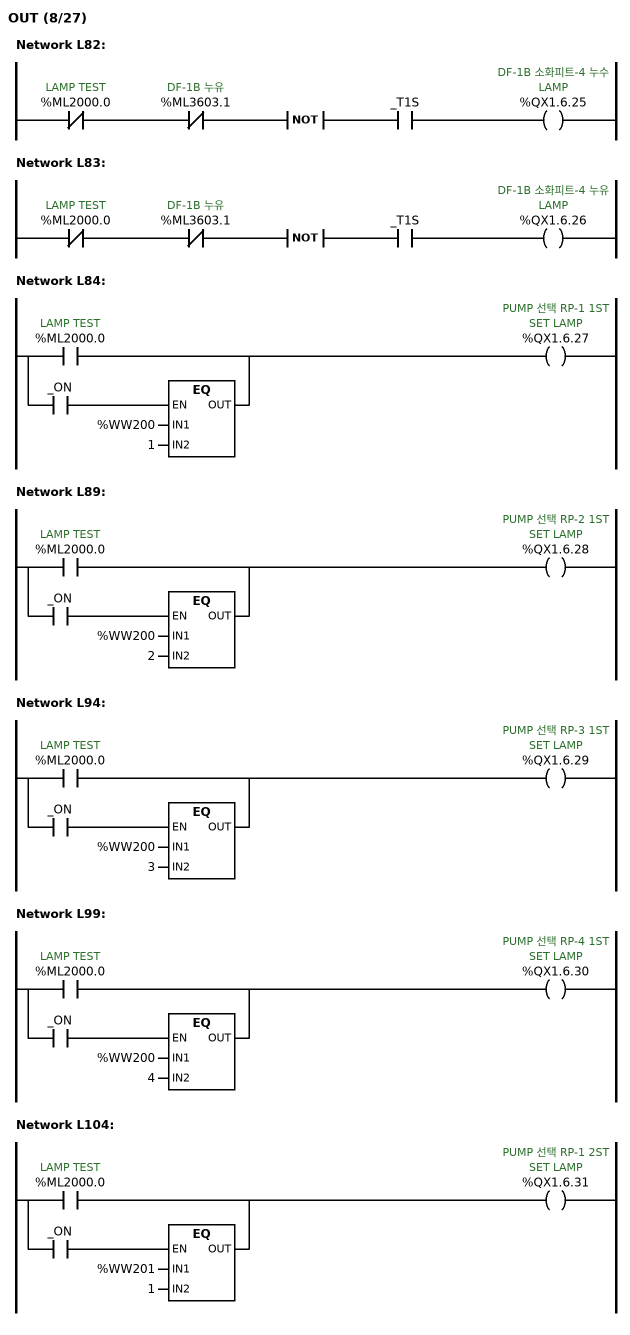
(* Rung L82 *)
%QX1.6.25 := NOT (NOT %ML2000.0 AND NOT %ML3603.1) AND _T1S;
(* Rung L83 *)
%QX1.6.26 := NOT (NOT %ML2000.0 AND NOT %ML3603.1) AND _T1S;
(* Rung L84 *)
IF _ON THEN _t1 := %WW200 = 1; END_IF;
%QX1.6.27 := %ML2000.0 OR _t1;
(* Rung L89 *)
IF _ON THEN _t2 := %WW200 = 2; END_IF;
%QX1.6.28 := %ML2000.0 OR _t2;
(* Rung L94 *)
IF _ON THEN _t3 := %WW200 = 3; END_IF;
%QX1.6.29 := %ML2000.0 OR _t3;
(* Rung L99 *)
IF _ON THEN _t4 := %WW200 = 4; END_IF;
%QX1.6.30 := %ML2000.0 OR _t4;
(* Rung L104 *)
IF _ON THEN _t5 := %WW201 = 1; END_IF;
%QX1.6.31 := %ML2000.0 OR _t5;

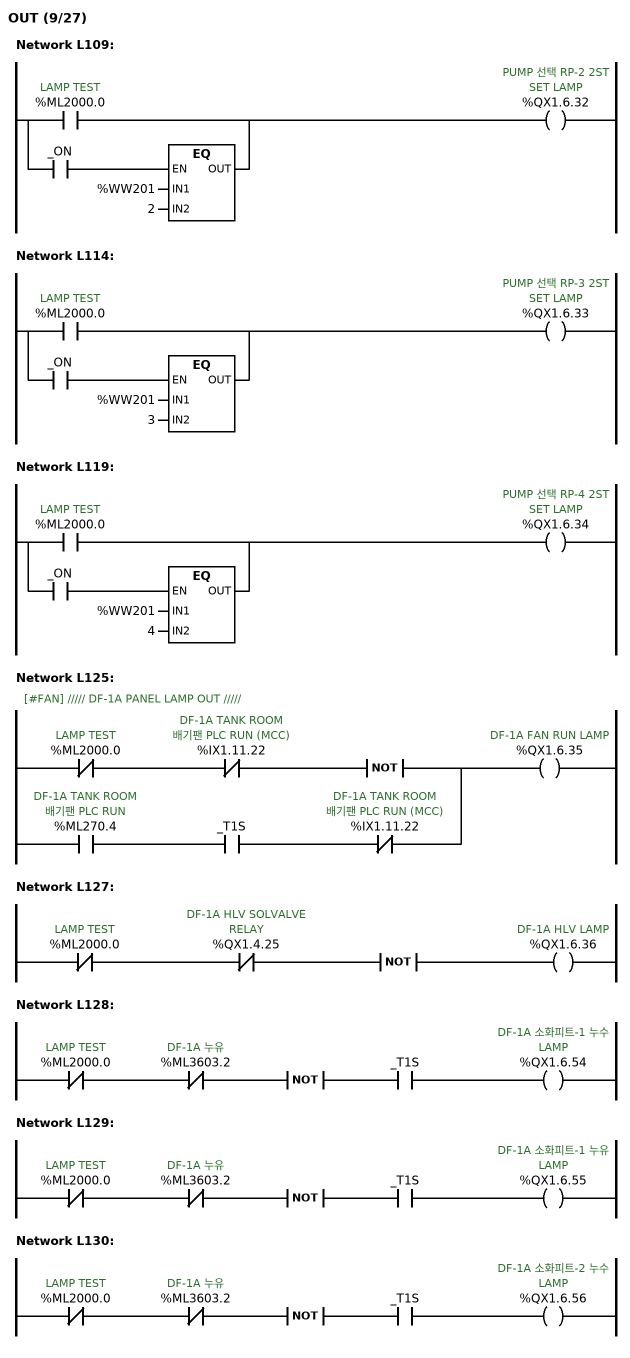
(* Rung L109 *)
IF _ON THEN _t6 := %WW201 = 2; END_IF;
%QX1.6.32 := %ML2000.0 OR _t6;
(* Rung L114 *)
IF _ON THEN _t7 := %WW201 = 3; END_IF;
%QX1.6.33 := %ML2000.0 OR _t7;
(* Rung L119 *)
IF _ON THEN _t8 := %WW201 = 4; END_IF;
%QX1.6.34 := %ML2000.0 OR _t8;
(* [#FAN] ///// DF-1A PANEL LAMP OUT ///// *)
(* Rung L125 *)
%QX1.6.35 := NOT (NOT %ML2000.0 AND NOT %IX1.11.22) OR (%ML270.4 AND _T1S AND NOT %IX1.11.22);
(* Rung L127 *)
%QX1.6.36 := NOT (NOT %ML2000.0 AND NOT %QX1.4.25);
(* Rung L128 *)
%QX1.6.54 := NOT (NOT %ML2000.0 AND NOT %ML3603.2) AND _T1S;
(* Rung L129 *)
%QX1.6.55 := NOT (NOT %ML2000.0 AND NOT %ML3603.2) AND _T1S;
(* Rung L130 *)
%QX1.6.56 := NOT (NOT %ML2000.0 AND NOT %ML3603.2) AND _T1S;

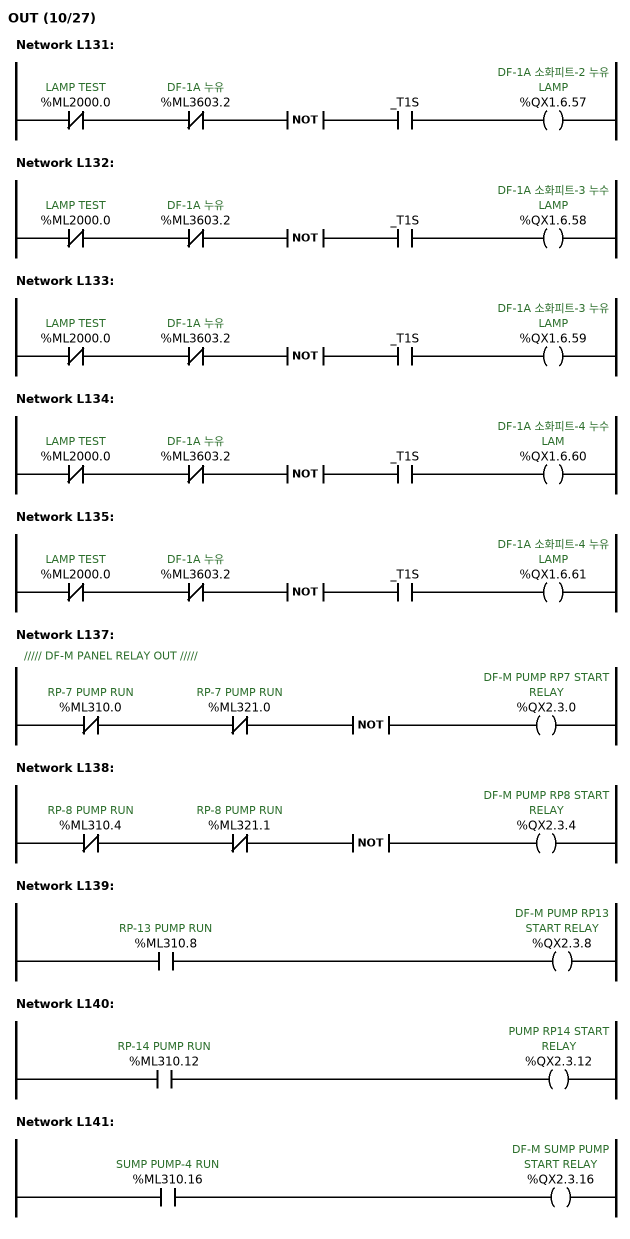
(* Rung L131 *)
%QX1.6.57 := NOT (NOT %ML2000.0 AND NOT %ML3603.2) AND _T1S;
(* Rung L132 *)
%QX1.6.58 := NOT (NOT %ML2000.0 AND NOT %ML3603.2) AND _T1S;
(* Rung L133 *)
%QX1.6.59 := NOT (NOT %ML2000.0 AND NOT %ML3603.2) AND _T1S;
(* Rung L134 *)
%QX1.6.60 := NOT (NOT %ML2000.0 AND NOT %ML3603.2) AND _T1S;
(* Rung L135 *)
%QX1.6.61 := NOT (NOT %ML2000.0 AND NOT %ML3603.2) AND _T1S;
(* ///// DF-M PANEL RELAY OUT ///// *)
(* Rung L137 *)
%QX2.3.0 := NOT (NOT %ML310.0 AND NOT %ML321.0);
(* Rung L138 *)
%QX2.3.4 := NOT (NOT %ML310.4 AND NOT %ML321.1);
(* Rung L139 *)
%QX2.3.8 := %ML310.8;
(* Rung L140 *)
%QX2.3.12 := %ML310.12;
(* Rung L141 *)
%QX2.3.16 := %ML310.16;

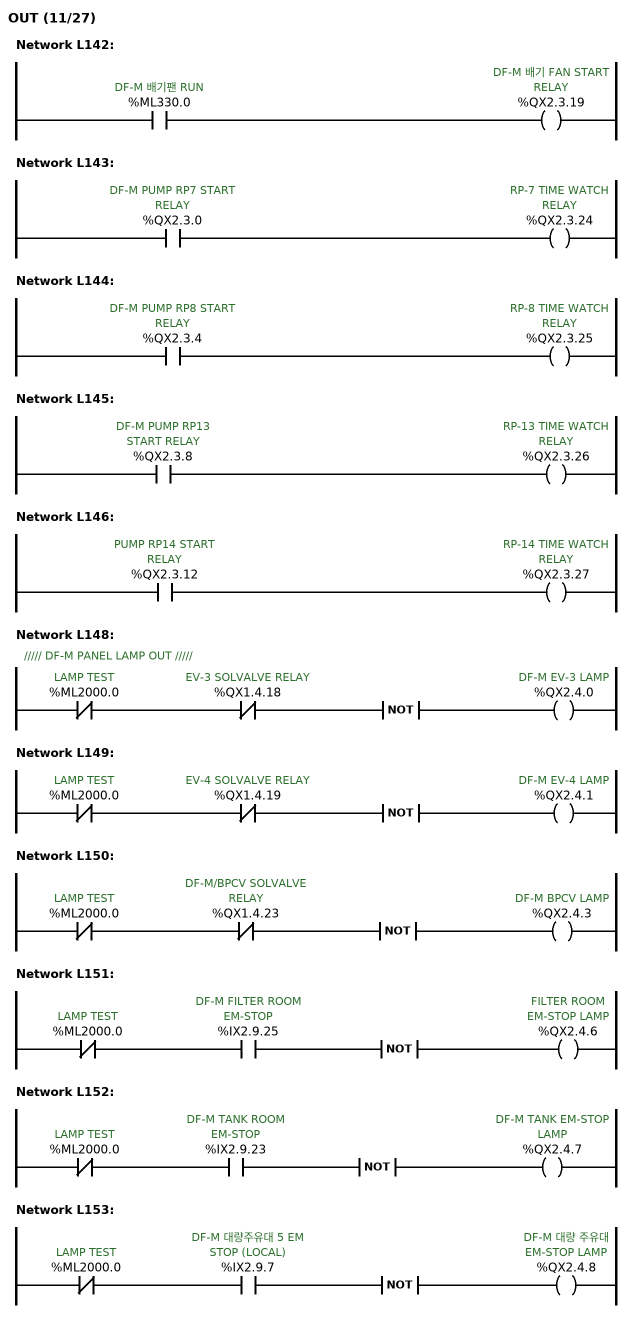
(* Rung L142 *)
%QX2.3.19 := %ML330.0;
(* Rung L143 *)
%QX2.3.24 := %QX2.3.0;
(* Rung L144 *)
%QX2.3.25 := %QX2.3.4;
(* Rung L145 *)
%QX2.3.26 := %QX2.3.8;
(* Rung L146 *)
%QX2.3.27 := %QX2.3.12;
(* ///// DF-M PANEL LAMP OUT ///// *)
(* Rung L148 *)
%QX2.4.0 := NOT (NOT %ML2000.0 AND NOT %QX1.4.18);
(* Rung L149 *)
%QX2.4.1 := NOT (NOT %ML2000.0 AND NOT %QX1.4.19);
(* Rung L150 *)
%QX2.4.3 := NOT (NOT %ML2000.0 AND NOT %QX1.4.23);
(* Rung L151 *)
%QX2.4.6 := NOT (NOT %ML2000.0 AND %IX2.9.25);
(* Rung L152 *)
%QX2.4.7 := NOT (NOT %ML2000.0 AND %IX2.9.23);
(* Rung L153 *)
%QX2.4.8 := NOT (NOT %ML2000.0 AND %IX2.9.7);

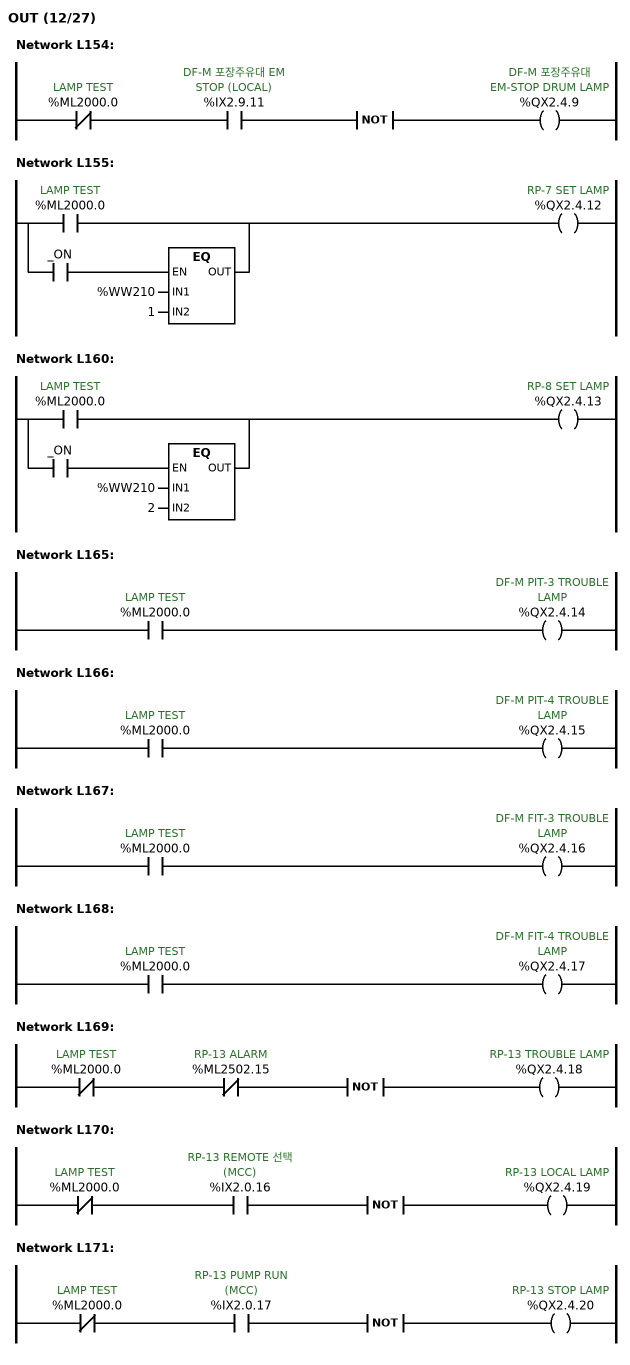
(* Rung L154 *)
%QX2.4.9 := NOT (NOT %ML2000.0 AND %IX2.9.11);
(* Rung L155 *)
IF _ON THEN _t9 := %WW210 = 1; END_IF;
%QX2.4.12 := %ML2000.0 OR _t9;
(* Rung L160 *)
IF _ON THEN _t10 := %WW210 = 2; END_IF;
%QX2.4.13 := %ML2000.0 OR _t10;
(* Rung L165 *)
%QX2.4.14 := %ML2000.0;
(* Rung L166 *)
%QX2.4.15 := %ML2000.0;
(* Rung L167 *)
%QX2.4.16 := %ML2000.0;
(* Rung L168 *)
%QX2.4.17 := %ML2000.0;
(* Rung L169 *)
%QX2.4.18 := NOT (NOT %ML2000.0 AND NOT %ML2502.15);
(* Rung L170 *)
%QX2.4.19 := NOT (NOT %ML2000.0 AND %IX2.0.16);
(* Rung L171 *)
%QX2.4.20 := NOT (NOT %ML2000.0 AND %IX2.0.17);

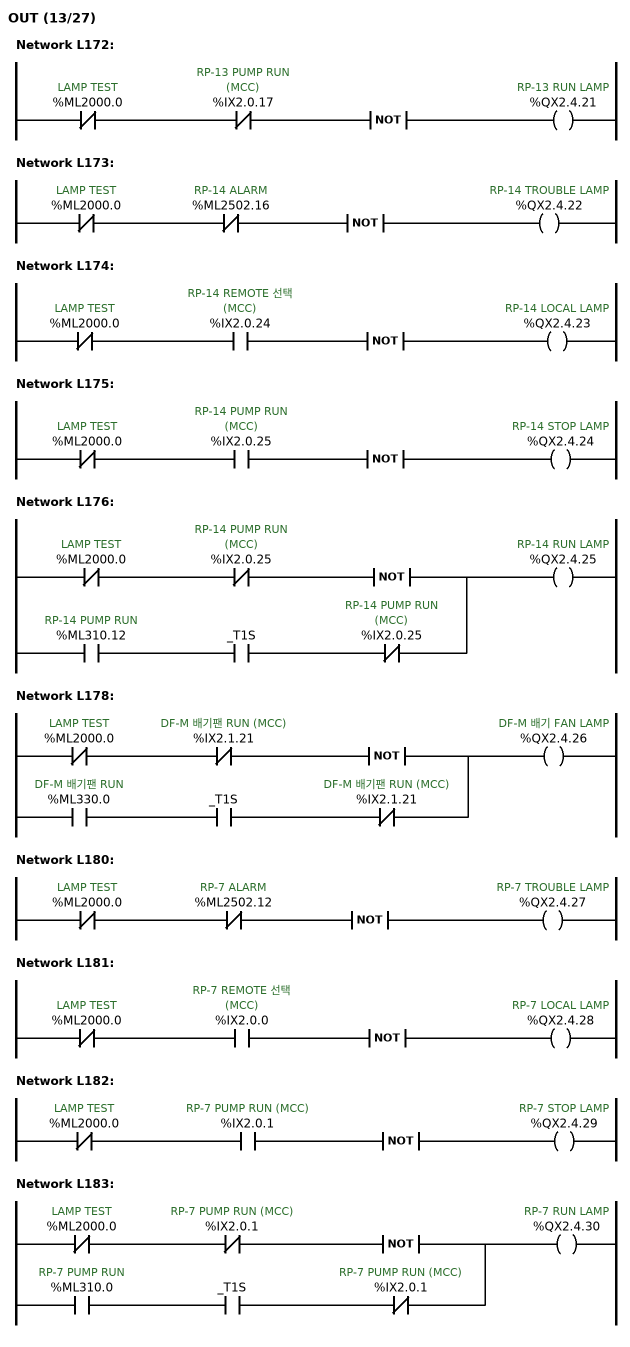
(* Rung L172 *)
%QX2.4.21 := NOT (NOT %ML2000.0 AND NOT %IX2.0.17);
(* Rung L173 *)
%QX2.4.22 := NOT (NOT %ML2000.0 AND NOT %ML2502.16);
(* Rung L174 *)
%QX2.4.23 := NOT (NOT %ML2000.0 AND %IX2.0.24);
(* Rung L175 *)
%QX2.4.24 := NOT (NOT %ML2000.0 AND %IX2.0.25);
(* Rung L176 *)
%QX2.4.25 := NOT (NOT %ML2000.0 AND NOT %IX2.0.25) OR (%ML310.12 AND _T1S AND NOT %IX2.0.25);
(* Rung L178 *)
%QX2.4.26 := NOT (NOT %ML2000.0 AND NOT %IX2.1.21) OR (%ML330.0 AND _T1S AND NOT %IX2.1.21);
(* Rung L180 *)
%QX2.4.27 := NOT (NOT %ML2000.0 AND NOT %ML2502.12);
(* Rung L181 *)
%QX2.4.28 := NOT (NOT %ML2000.0 AND %IX2.0.0);
(* Rung L182 *)
%QX2.4.29 := NOT (NOT %ML2000.0 AND %IX2.0.1);
(* Rung L183 *)
%QX2.4.30 := NOT (NOT %ML2000.0 AND NOT %IX2.0.1) OR (%ML310.0 AND _T1S AND NOT %IX2.0.1);

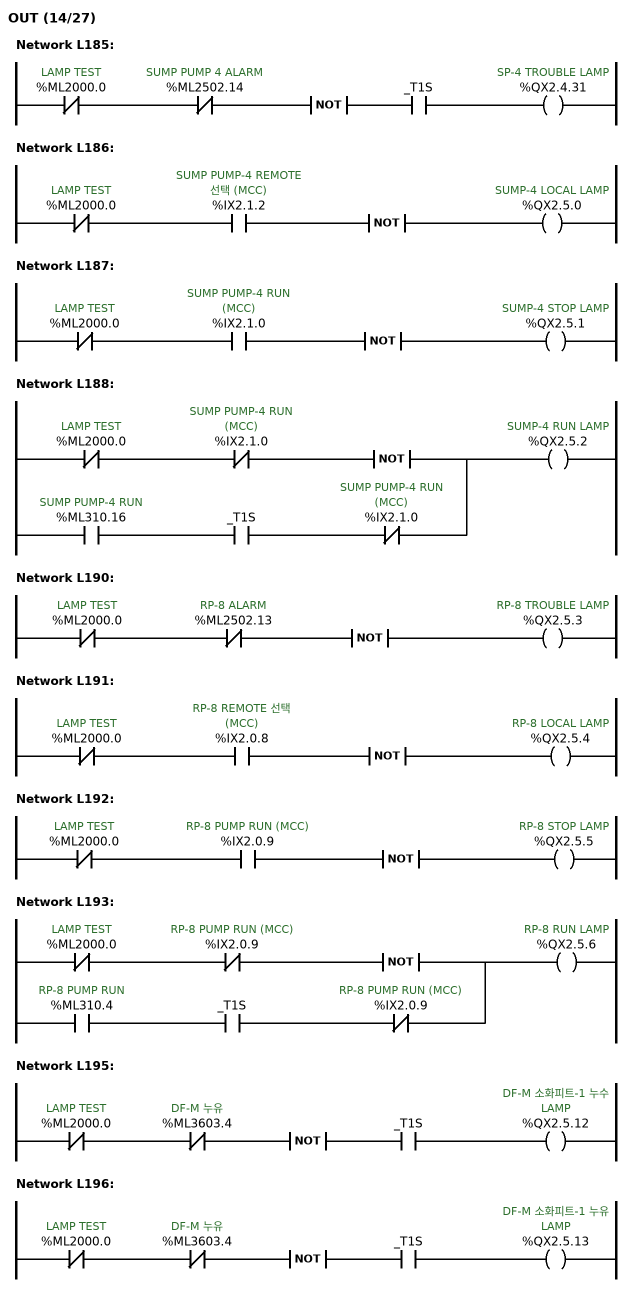
(* Rung L185 *)
%QX2.4.31 := NOT (NOT %ML2000.0 AND NOT %ML2502.14) AND _T1S;
(* Rung L186 *)
%QX2.5.0 := NOT (NOT %ML2000.0 AND %IX2.1.2);
(* Rung L187 *)
%QX2.5.1 := NOT (NOT %ML2000.0 AND %IX2.1.0);
(* Rung L188 *)
%QX2.5.2 := NOT (NOT %ML2000.0 AND NOT %IX2.1.0) OR (%ML310.16 AND _T1S AND NOT %IX2.1.0);
(* Rung L190 *)
%QX2.5.3 := NOT (NOT %ML2000.0 AND NOT %ML2502.13);
(* Rung L191 *)
%QX2.5.4 := NOT (NOT %ML2000.0 AND %IX2.0.8);
(* Rung L192 *)
%QX2.5.5 := NOT (NOT %ML2000.0 AND %IX2.0.9);
(* Rung L193 *)
%QX2.5.6 := NOT (NOT %ML2000.0 AND NOT %IX2.0.9) OR (%ML310.4 AND _T1S AND NOT %IX2.0.9);
(* Rung L195 *)
%QX2.5.12 := NOT (NOT %ML2000.0 AND NOT %ML3603.4) AND _T1S;
(* Rung L196 *)
%QX2.5.13 := NOT (NOT %ML2000.0 AND NOT %ML3603.4) AND _T1S;

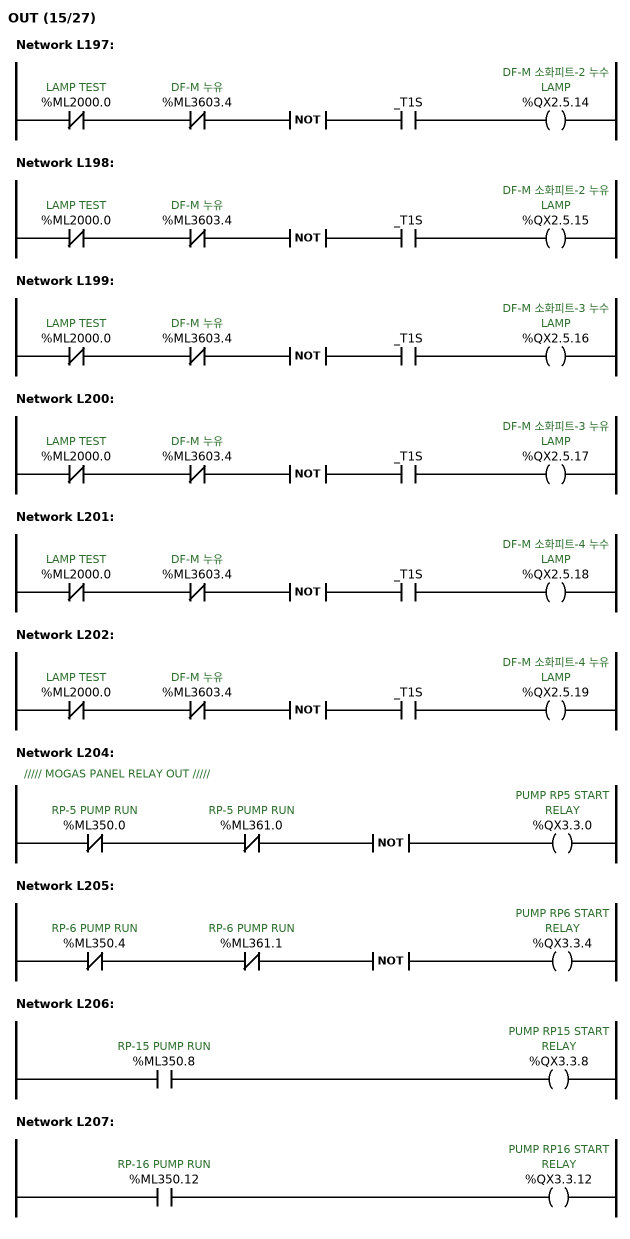
(* Rung L197 *)
%QX2.5.14 := NOT (NOT %ML2000.0 AND NOT %ML3603.4) AND _T1S;
(* Rung L198 *)
%QX2.5.15 := NOT (NOT %ML2000.0 AND NOT %ML3603.4) AND _T1S;
(* Rung L199 *)
%QX2.5.16 := NOT (NOT %ML2000.0 AND NOT %ML3603.4) AND _T1S;
(* Rung L200 *)
%QX2.5.17 := NOT (NOT %ML2000.0 AND NOT %ML3603.4) AND _T1S;
(* Rung L201 *)
%QX2.5.18 := NOT (NOT %ML2000.0 AND NOT %ML3603.4) AND _T1S;
(* Rung L202 *)
%QX2.5.19 := NOT (NOT %ML2000.0 AND NOT %ML3603.4) AND _T1S;
(* ///// MOGAS PANEL RELAY OUT ///// *)
(* Rung L204 *)
%QX3.3.0 := NOT (NOT %ML350.0 AND NOT %ML361.0);
(* Rung L205 *)
%QX3.3.4 := NOT (NOT %ML350.4 AND NOT %ML361.1);
(* Rung L206 *)
%QX3.3.8 := %ML350.8;
(* Rung L207 *)
%QX3.3.12 := %ML350.12;

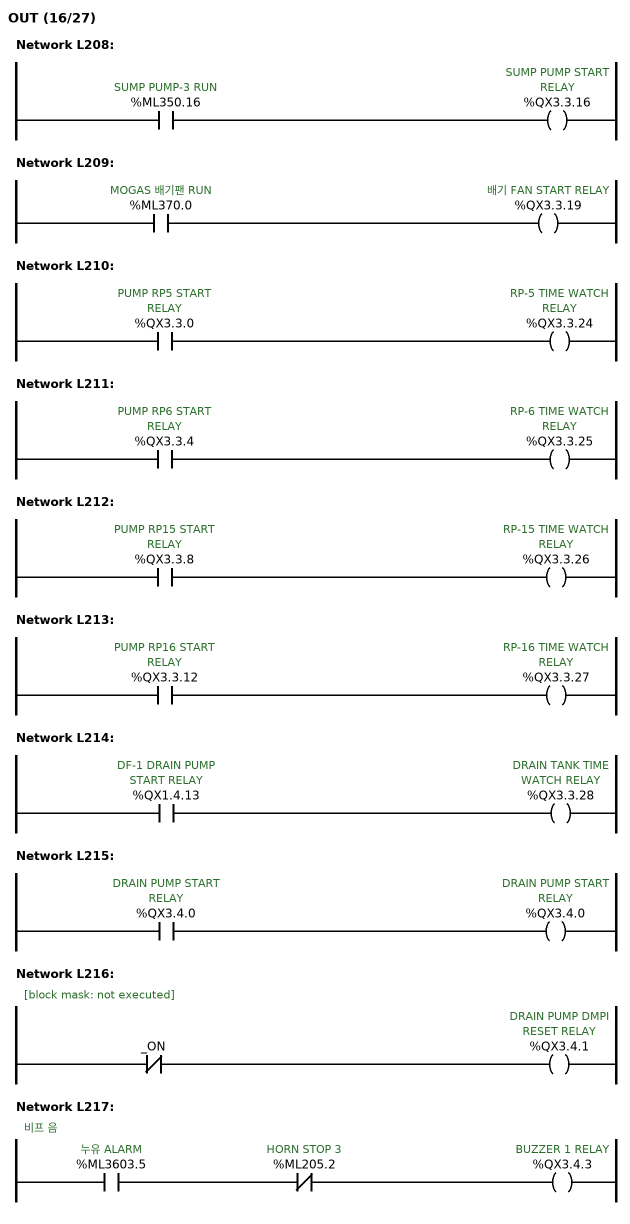
(* Rung L208 *)
%QX3.3.16 := %ML350.16;
(* Rung L209 *)
%QX3.3.19 := %ML370.0;
(* Rung L210 *)
%QX3.3.24 := %QX3.3.0;
(* Rung L211 *)
%QX3.3.25 := %QX3.3.4;
(* Rung L212 *)
%QX3.3.26 := %QX3.3.8;
(* Rung L213 *)
%QX3.3.27 := %QX3.3.12;
(* Rung L214 *)
%QX3.3.28 := %QX1.4.13;
(* Rung L215 *)
%QX3.4.0 := %QX3.4.0;
(* Rung L216 is block-masked: not executed *)
// %QX3.4.1 := NOT _ON;
(* Rung L217 *)
%QX3.4.3 := %ML3603.5 AND NOT %ML205.2;
(* 비프 음 *)

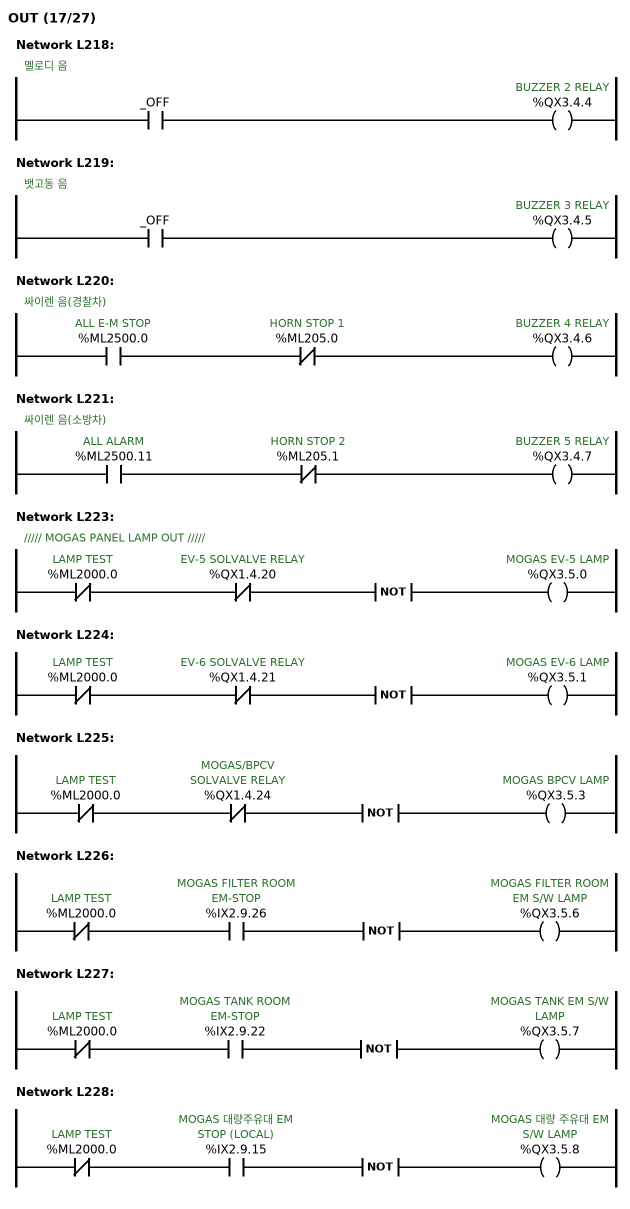
(* Rung L218 *)
%QX3.4.4 := _OFF;
(* 멜로디 음 *)
(* Rung L219 *)
%QX3.4.5 := _OFF;
(* 뱃고동 음 *)
(* Rung L220 *)
%QX3.4.6 := %ML2500.0 AND NOT %ML205.0;
(* 싸이렌 음(경찰차) *)
(* Rung L221 *)
%QX3.4.7 := %ML2500.11 AND NOT %ML205.1;
(* 싸이렌 음(소방차) *)
(* ///// MOGAS PANEL LAMP OUT ///// *)
(* Rung L223 *)
%QX3.5.0 := NOT (NOT %ML2000.0 AND NOT %QX1.4.20);
(* Rung L224 *)
%QX3.5.1 := NOT (NOT %ML2000.0 AND NOT %QX1.4.21);
(* Rung L225 *)
%QX3.5.3 := NOT (NOT %ML2000.0 AND NOT %QX1.4.24);
(* Rung L226 *)
%QX3.5.6 := NOT (NOT %ML2000.0 AND %IX2.9.26);
(* Rung L227 *)
%QX3.5.7 := NOT (NOT %ML2000.0 AND %IX2.9.22);
(* Rung L228 *)
%QX3.5.8 := NOT (NOT %ML2000.0 AND %IX2.9.15);

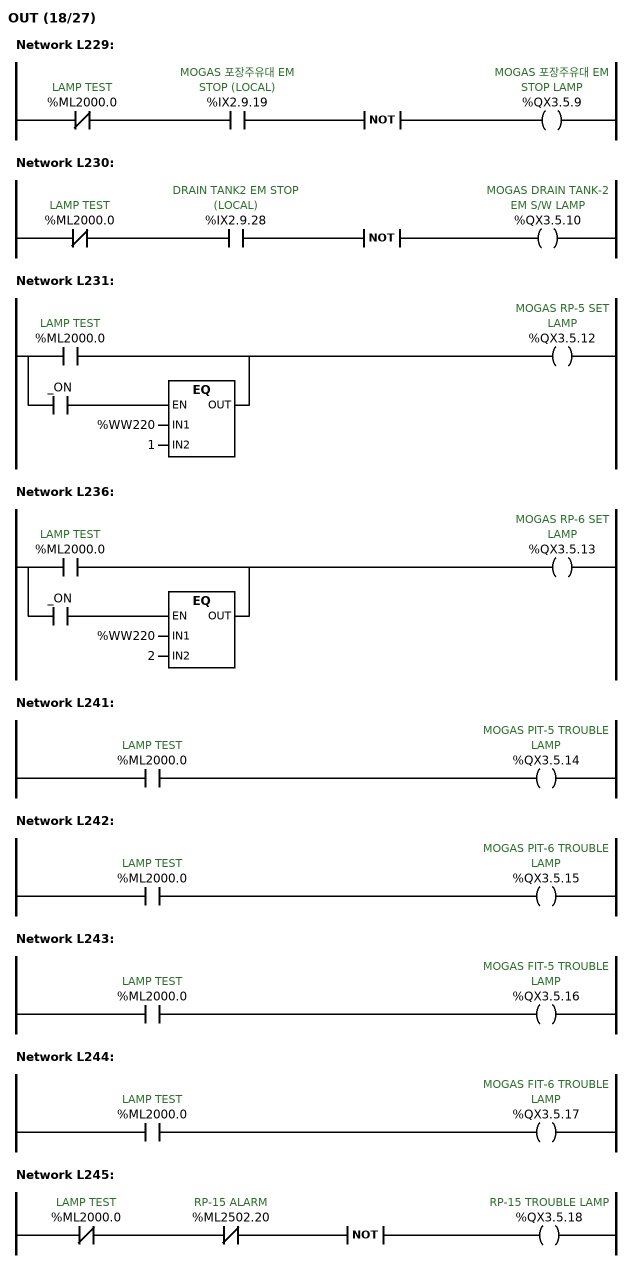
(* Rung L229 *)
%QX3.5.9 := NOT (NOT %ML2000.0 AND %IX2.9.19);
(* Rung L230 *)
%QX3.5.10 := NOT (NOT %ML2000.0 AND %IX2.9.28);
(* Rung L231 *)
IF _ON THEN _t11 := %WW220 = 1; END_IF;
%QX3.5.12 := %ML2000.0 OR _t11;
(* Rung L236 *)
IF _ON THEN _t12 := %WW220 = 2; END_IF;
%QX3.5.13 := %ML2000.0 OR _t12;
(* Rung L241 *)
%QX3.5.14 := %ML2000.0;
(* Rung L242 *)
%QX3.5.15 := %ML2000.0;
(* Rung L243 *)
%QX3.5.16 := %ML2000.0;
(* Rung L244 *)
%QX3.5.17 := %ML2000.0;
(* Rung L245 *)
%QX3.5.18 := NOT (NOT %ML2000.0 AND NOT %ML2502.20);

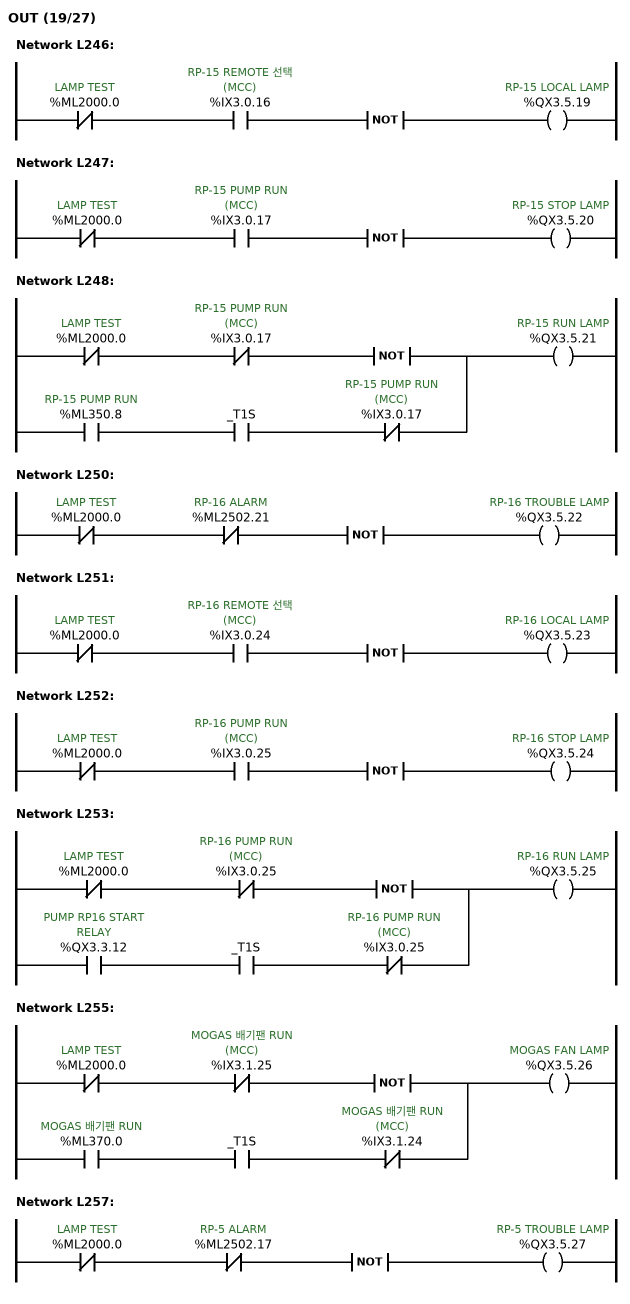
(* Rung L246 *)
%QX3.5.19 := NOT (NOT %ML2000.0 AND %IX3.0.16);
(* Rung L247 *)
%QX3.5.20 := NOT (NOT %ML2000.0 AND %IX3.0.17);
(* Rung L248 *)
%QX3.5.21 := NOT (NOT %ML2000.0 AND NOT %IX3.0.17) OR (%ML350.8 AND _T1S AND NOT %IX3.0.17);
(* Rung L250 *)
%QX3.5.22 := NOT (NOT %ML2000.0 AND NOT %ML2502.21);
(* Rung L251 *)
%QX3.5.23 := NOT (NOT %ML2000.0 AND %IX3.0.24);
(* Rung L252 *)
%QX3.5.24 := NOT (NOT %ML2000.0 AND %IX3.0.25);
(* Rung L253 *)
%QX3.5.25 := NOT (NOT %ML2000.0 AND NOT %IX3.0.25) OR (%QX3.3.12 AND _T1S AND NOT %IX3.0.25);
(* Rung L255 *)
%QX3.5.26 := NOT (NOT %ML2000.0 AND NOT %IX3.1.25) OR (%ML370.0 AND _T1S AND NOT %IX3.1.24);
(* Rung L257 *)
%QX3.5.27 := NOT (NOT %ML2000.0 AND NOT %ML2502.17);

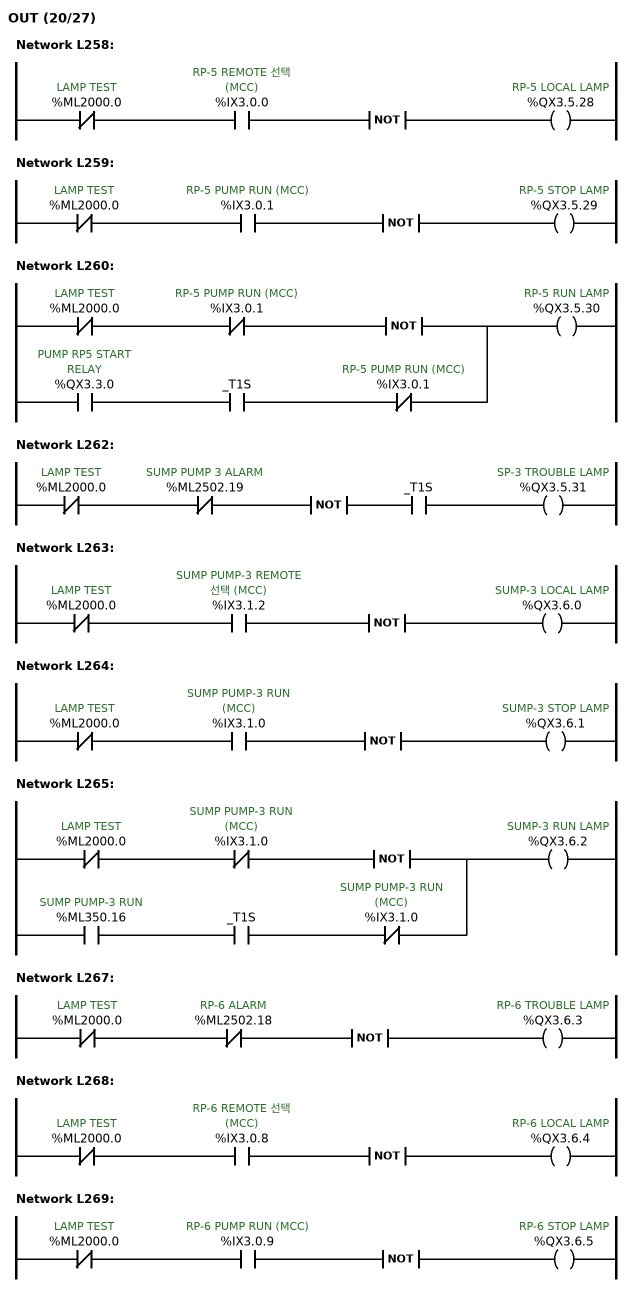
(* Rung L258 *)
%QX3.5.28 := NOT (NOT %ML2000.0 AND %IX3.0.0);
(* Rung L259 *)
%QX3.5.29 := NOT (NOT %ML2000.0 AND %IX3.0.1);
(* Rung L260 *)
%QX3.5.30 := NOT (NOT %ML2000.0 AND NOT %IX3.0.1) OR (%QX3.3.0 AND _T1S AND NOT %IX3.0.1);
(* Rung L262 *)
%QX3.5.31 := NOT (NOT %ML2000.0 AND NOT %ML2502.19) AND _T1S;
(* Rung L263 *)
%QX3.6.0 := NOT (NOT %ML2000.0 AND %IX3.1.2);
(* Rung L264 *)
%QX3.6.1 := NOT (NOT %ML2000.0 AND %IX3.1.0);
(* Rung L265 *)
%QX3.6.2 := NOT (NOT %ML2000.0 AND NOT %IX3.1.0) OR (%ML350.16 AND _T1S AND NOT %IX3.1.0);
(* Rung L267 *)
%QX3.6.3 := NOT (NOT %ML2000.0 AND NOT %ML2502.18);
(* Rung L268 *)
%QX3.6.4 := NOT (NOT %ML2000.0 AND %IX3.0.8);
(* Rung L269 *)
%QX3.6.5 := NOT (NOT %ML2000.0 AND %IX3.0.9);

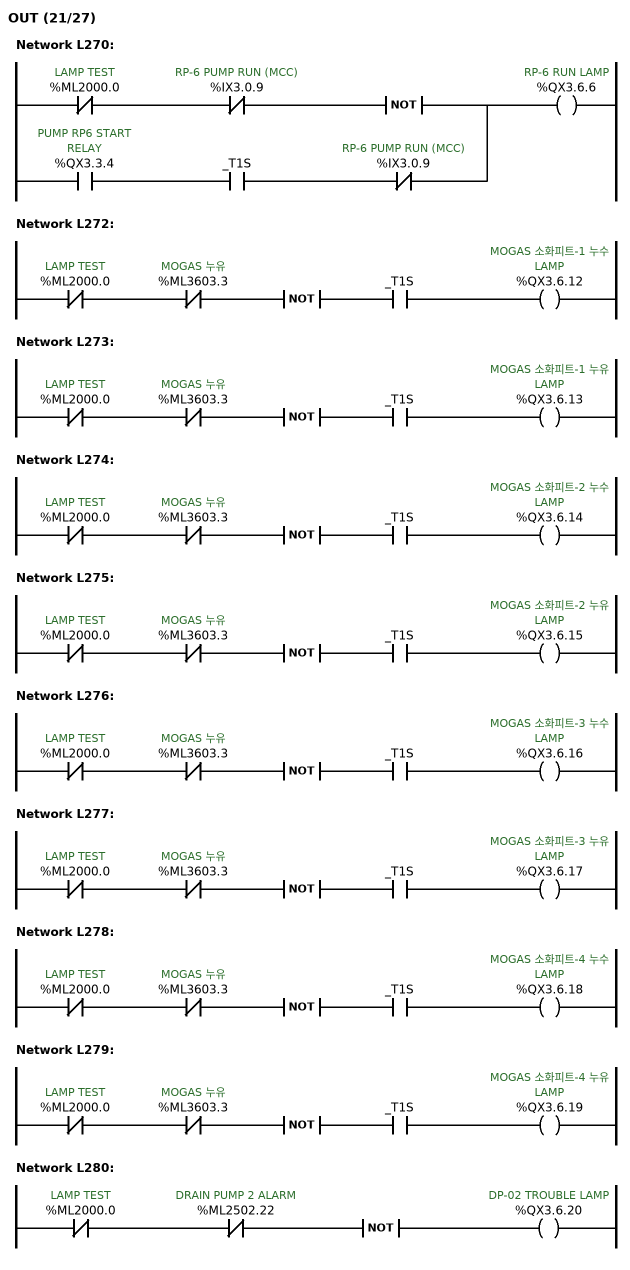
(* Rung L270 *)
%QX3.6.6 := NOT (NOT %ML2000.0 AND NOT %IX3.0.9) OR (%QX3.3.4 AND _T1S AND NOT %IX3.0.9);
(* Rung L272 *)
%QX3.6.12 := NOT (NOT %ML2000.0 AND NOT %ML3603.3) AND _T1S;
(* Rung L273 *)
%QX3.6.13 := NOT (NOT %ML2000.0 AND NOT %ML3603.3) AND _T1S;
(* Rung L274 *)
%QX3.6.14 := NOT (NOT %ML2000.0 AND NOT %ML3603.3) AND _T1S;
(* Rung L275 *)
%QX3.6.15 := NOT (NOT %ML2000.0 AND NOT %ML3603.3) AND _T1S;
(* Rung L276 *)
%QX3.6.16 := NOT (NOT %ML2000.0 AND NOT %ML3603.3) AND _T1S;
(* Rung L277 *)
%QX3.6.17 := NOT (NOT %ML2000.0 AND NOT %ML3603.3) AND _T1S;
(* Rung L278 *)
%QX3.6.18 := NOT (NOT %ML2000.0 AND NOT %ML3603.3) AND _T1S;
(* Rung L279 *)
%QX3.6.19 := NOT (NOT %ML2000.0 AND NOT %ML3603.3) AND _T1S;
(* Rung L280 *)
%QX3.6.20 := NOT (NOT %ML2000.0 AND NOT %ML2502.22);

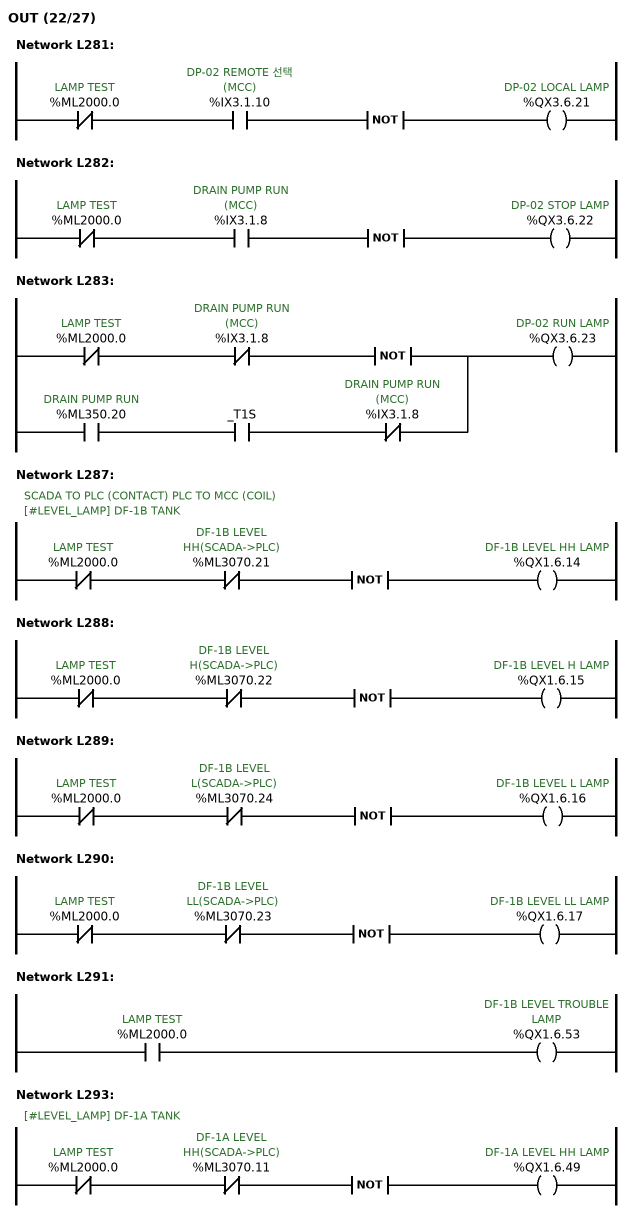
(* Rung L281 *)
%QX3.6.21 := NOT (NOT %ML2000.0 AND %IX3.1.10);
(* Rung L282 *)
%QX3.6.22 := NOT (NOT %ML2000.0 AND %IX3.1.8);
(* Rung L283 *)
%QX3.6.23 := NOT (NOT %ML2000.0 AND NOT %IX3.1.8) OR (%ML350.20 AND _T1S AND NOT %IX3.1.8);
(* SCADA TO PLC (CONTACT) PLC TO MCC (COIL) *)
(* [#LEVEL_LAMP] DF-1B TANK *)
(* Rung L287 *)
%QX1.6.14 := NOT (NOT %ML2000.0 AND NOT %ML3070.21);
(* Rung L288 *)
%QX1.6.15 := NOT (NOT %ML2000.0 AND NOT %ML3070.22);
(* Rung L289 *)
%QX1.6.16 := NOT (NOT %ML2000.0 AND NOT %ML3070.24);
(* Rung L290 *)
%QX1.6.17 := NOT (NOT %ML2000.0 AND NOT %ML3070.23);
(* Rung L291 *)
%QX1.6.53 := %ML2000.0;
(* [#LEVEL_LAMP] DF-1A TANK *)
(* Rung L293 *)
%QX1.6.49 := NOT (NOT %ML2000.0 AND NOT %ML3070.11);

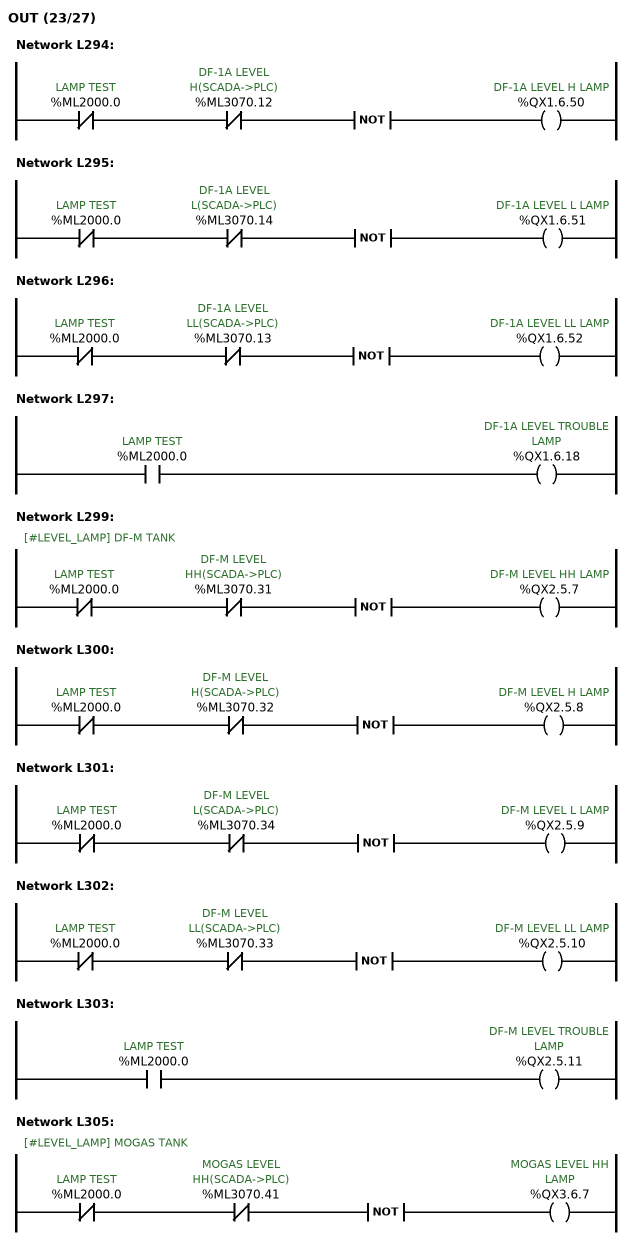
(* Rung L294 *)
%QX1.6.50 := NOT (NOT %ML2000.0 AND NOT %ML3070.12);
(* Rung L295 *)
%QX1.6.51 := NOT (NOT %ML2000.0 AND NOT %ML3070.14);
(* Rung L296 *)
%QX1.6.52 := NOT (NOT %ML2000.0 AND NOT %ML3070.13);
(* Rung L297 *)
%QX1.6.18 := %ML2000.0;
(* [#LEVEL_LAMP] DF-M TANK *)
(* Rung L299 *)
%QX2.5.7 := NOT (NOT %ML2000.0 AND NOT %ML3070.31);
(* Rung L300 *)
%QX2.5.8 := NOT (NOT %ML2000.0 AND NOT %ML3070.32);
(* Rung L301 *)
%QX2.5.9 := NOT (NOT %ML2000.0 AND NOT %ML3070.34);
(* Rung L302 *)
%QX2.5.10 := NOT (NOT %ML2000.0 AND NOT %ML3070.33);
(* Rung L303 *)
%QX2.5.11 := %ML2000.0;
(* [#LEVEL_LAMP] MOGAS TANK *)
(* Rung L305 *)
%QX3.6.7 := NOT (NOT %ML2000.0 AND NOT %ML3070.41);

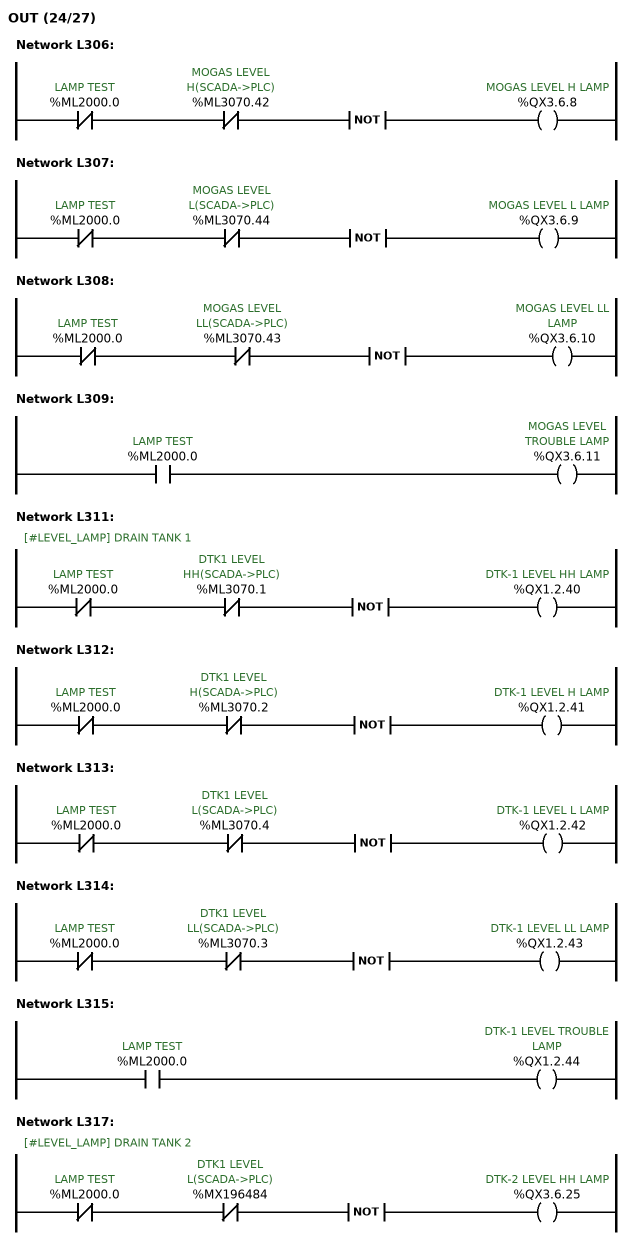
(* Rung L306 *)
%QX3.6.8 := NOT (NOT %ML2000.0 AND NOT %ML3070.42);
(* Rung L307 *)
%QX3.6.9 := NOT (NOT %ML2000.0 AND NOT %ML3070.44);
(* Rung L308 *)
%QX3.6.10 := NOT (NOT %ML2000.0 AND NOT %ML3070.43);
(* Rung L309 *)
%QX3.6.11 := %ML2000.0;
(* [#LEVEL_LAMP] DRAIN TANK 1 *)
(* Rung L311 *)
%QX1.2.40 := NOT (NOT %ML2000.0 AND NOT %ML3070.1);
(* Rung L312 *)
%QX1.2.41 := NOT (NOT %ML2000.0 AND NOT %ML3070.2);
(* Rung L313 *)
%QX1.2.42 := NOT (NOT %ML2000.0 AND NOT %ML3070.4);
(* Rung L314 *)
%QX1.2.43 := NOT (NOT %ML2000.0 AND NOT %ML3070.3);
(* Rung L315 *)
%QX1.2.44 := %ML2000.0;
(* [#LEVEL_LAMP] DRAIN TANK 2 *)
(* Rung L317 *)
%QX3.6.25 := NOT (NOT %ML2000.0 AND NOT %MX196484);

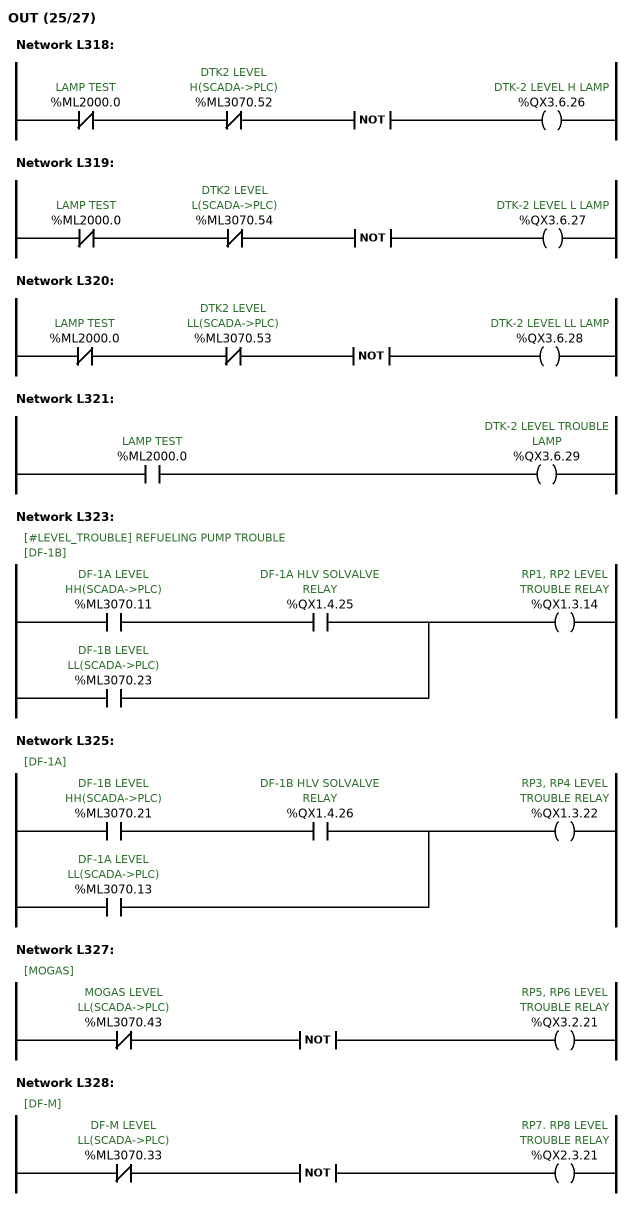
(* Rung L318 *)
%QX3.6.26 := NOT (NOT %ML2000.0 AND NOT %ML3070.52);
(* Rung L319 *)
%QX3.6.27 := NOT (NOT %ML2000.0 AND NOT %ML3070.54);
(* Rung L320 *)
%QX3.6.28 := NOT (NOT %ML2000.0 AND NOT %ML3070.53);
(* Rung L321 *)
%QX3.6.29 := %ML2000.0;
(* [#LEVEL_TROUBLE] REFUELING PUMP TROUBLE *)
(* Rung L323 *)
%QX1.3.14 := (%ML3070.11 AND %QX1.4.25) OR %ML3070.23;
(* [DF-1B] *)
(* Rung L325 *)
%QX1.3.22 := (%ML3070.21 AND %QX1.4.26) OR %ML3070.13;
(* [DF-1A] *)
(* Rung L327 *)
%QX3.2.21 := %ML3070.43;
(* [MOGAS] *)
(* Rung L328 *)
%QX2.3.21 := %ML3070.33;
(* [DF-M] *)

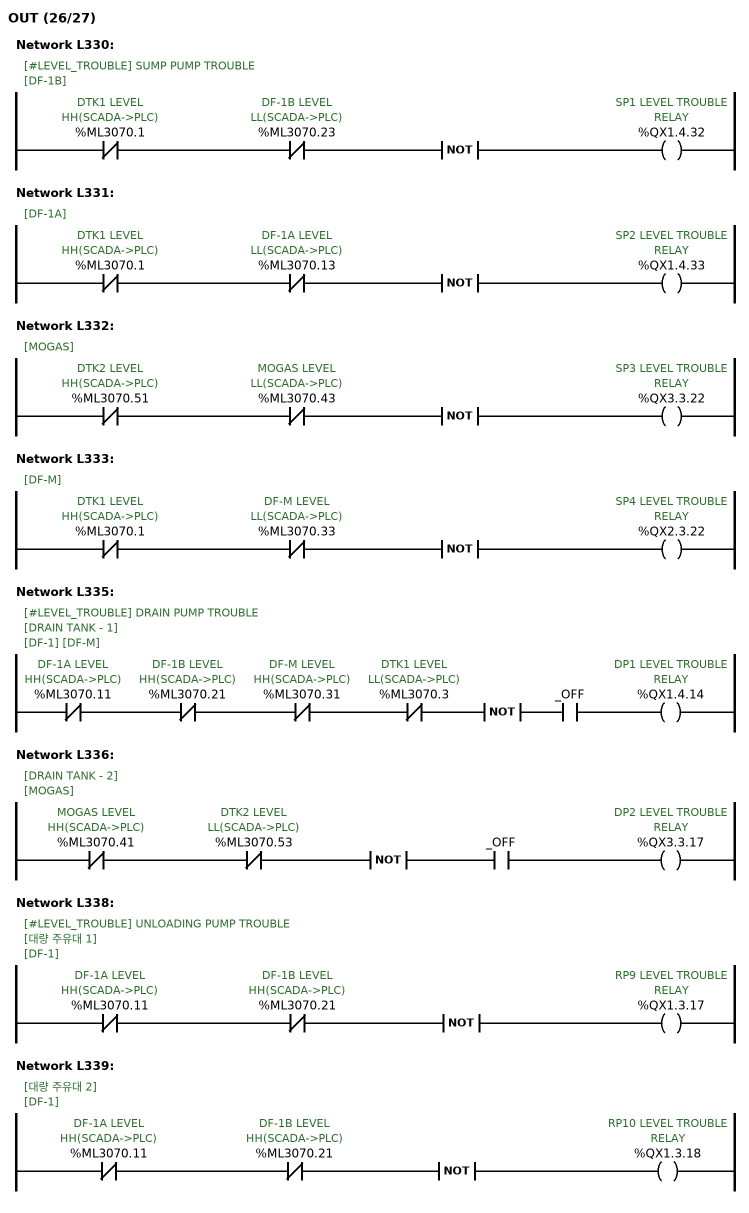
(* [#LEVEL_TROUBLE] SUMP PUMP TROUBLE *)
(* Rung L330 *)
%QX1.4.32 := NOT (NOT %ML3070.1 AND NOT %ML3070.23);
(* [DF-1B] *)
(* Rung L331 *)
%QX1.4.33 := NOT (NOT %ML3070.1 AND NOT %ML3070.13);
(* [DF-1A] *)
(* Rung L332 *)
%QX3.3.22 := NOT (NOT %ML3070.51 AND NOT %ML3070.43);
(* [MOGAS] *)
(* Rung L333 *)
%QX2.3.22 := NOT (NOT %ML3070.1 AND NOT %ML3070.33);
(* [DF-M] *)
(* [#LEVEL_TROUBLE] DRAIN PUMP TROUBLE *)
(* Rung L335 *)
%QX1.4.14 := NOT (NOT %ML3070.11 AND NOT %ML3070.21 AND NOT %ML3070.31 AND NOT %ML3070.3) AND _OFF;
(* [DRAIN TANK - 1] / [DF-1] [DF-M] *)
(* Rung L336 *)
%QX3.3.17 := NOT (NOT %ML3070.41 AND NOT %ML3070.53) AND _OFF;
(* [DRAIN TANK - 2] / [MOGAS] *)
(* [#LEVEL_TROUBLE] UNLOADING PUMP TROUBLE *)
(* Rung L338 *)
%QX1.3.17 := NOT (NOT %ML3070.11 AND NOT %ML3070.21);
(* [대량 주유대 1] / [DF-1] *)
(* Rung L339 *)
%QX1.3.18 := NOT (NOT %ML3070.11 AND NOT %ML3070.21);
(* [대량 주유대 2] / [DF-1] *)

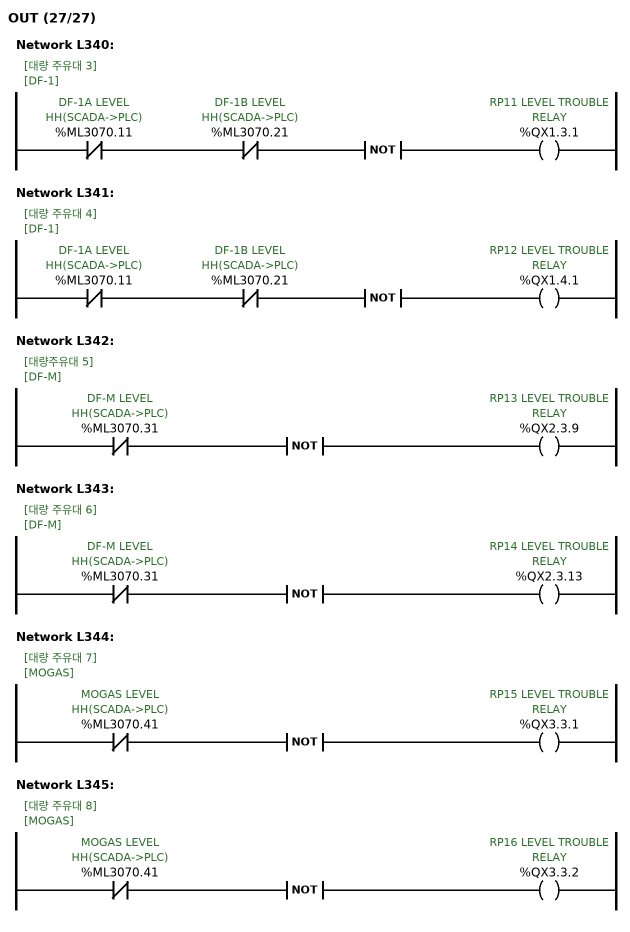
(* Rung L340 *)
%QX1.3.1 := NOT (NOT %ML3070.11 AND NOT %ML3070.21);
(* [대량 주유대 3] / [DF-1] *)
(* Rung L341 *)
%QX1.4.1 := NOT (NOT %ML3070.11 AND NOT %ML3070.21);
(* [대량 주유대 4] / [DF-1] *)
(* Rung L342 *)
%QX2.3.9 := %ML3070.31;
(* [대량주유대 5] / [DF-M] *)
(* Rung L343 *)
%QX2.3.13 := %ML3070.31;
(* [대량 주유대 6] / [DF-M] *)
(* Rung L344 *)
%QX3.3.1 := %ML3070.41;
(* [대량 주유대 7] / [MOGAS] *)
(* Rung L345 *)
%QX3.3.2 := %ML3070.41;
(* [대량 주유대 8] / [MOGAS] *)
END_PROGRAM

PROGRAM ALARM (* task: 스캔 프로그램 *)

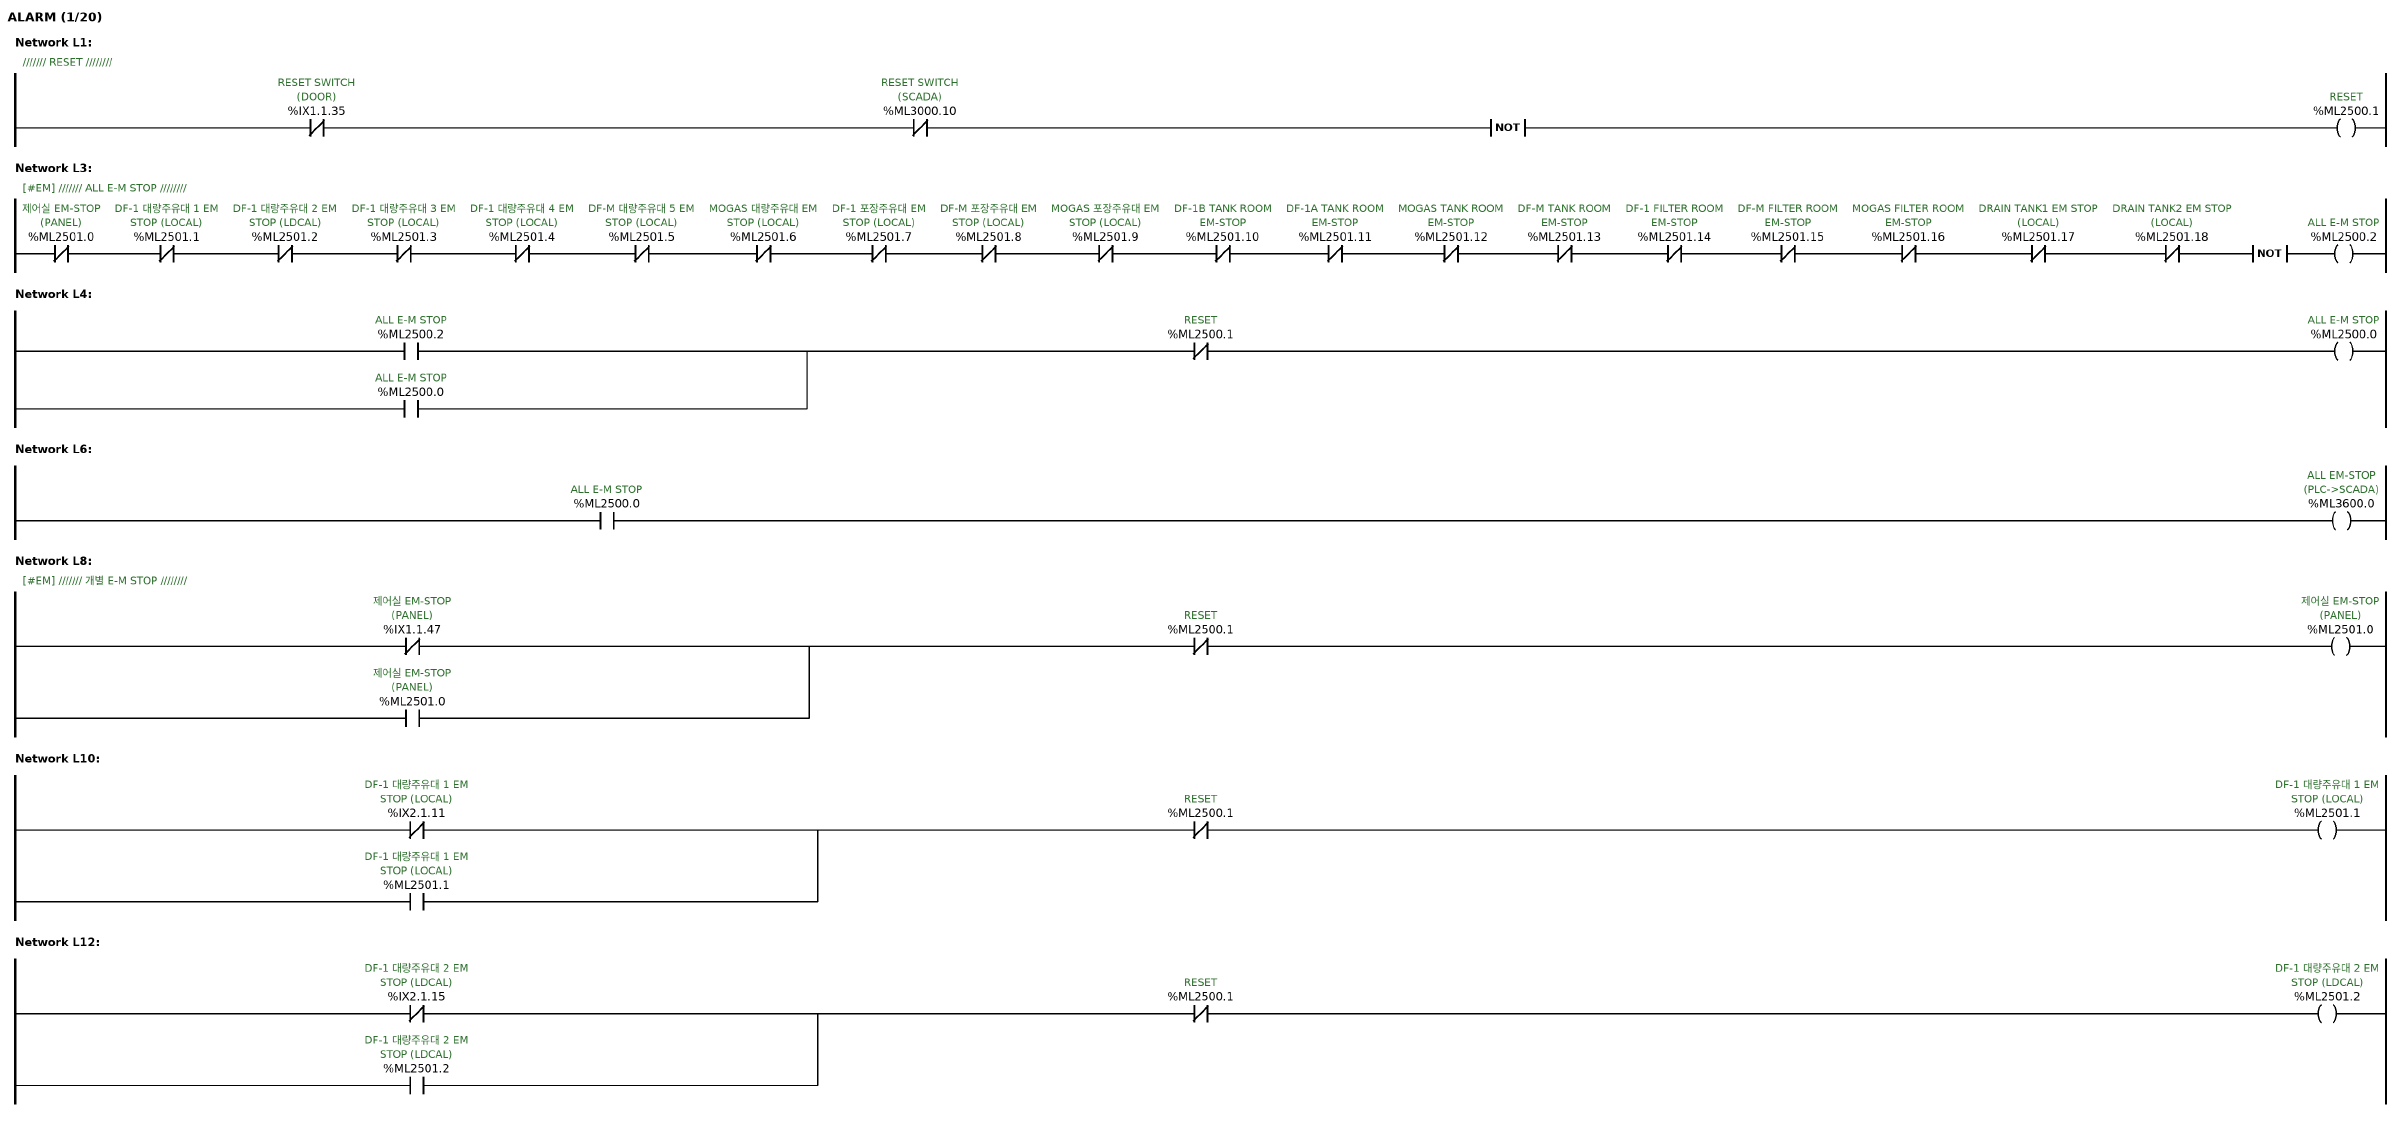
(* /////// RESET //////// *)
(* Rung L1 *)
%ML2500.1 := NOT (NOT %IX1.1.35 AND NOT %ML3000.10);
(* [#EM] /////// ALL E-M STOP //////// *)
(* Rung L3 *)
%ML2500.2 := NOT (NOT %ML2501.0 AND NOT %ML2501.1 AND NOT %ML2501.2 AND NOT %ML2501.3 AND NOT %ML2501.4 AND NOT %ML2501.5 AND NOT %ML2501.6 AND NOT %ML2501.7 AND NOT %ML2501.8 AND NOT %ML2501.9 AND NOT %ML2501.10 AND NOT %ML2501.11 AND NOT %ML2501.12 AND NOT %ML2501.13 AND NOT %ML2501.14 AND NOT %ML2501.15 AND NOT %ML2501.16 AND NOT %ML2501.17 AND NOT %ML2501.18);
(* Rung L4 *)
%ML2500.0 := (%ML2500.2 OR %ML2500.0) AND NOT %ML2500.1;
(* Rung L6 *)
%ML3600.0 := %ML2500.0;
(* [#EM] /////// 개별 E-M STOP //////// *)
(* Rung L8 *)
%ML2501.0 := (NOT %IX1.1.47 OR %ML2501.0) AND NOT %ML2500.1;
(* Rung L10 *)
%ML2501.1 := (NOT %IX2.1.11 OR %ML2501.1) AND NOT %ML2500.1;
(* Rung L12 *)
%ML2501.2 := (NOT %IX2.1.15 OR %ML2501.2) AND NOT %ML2500.1;

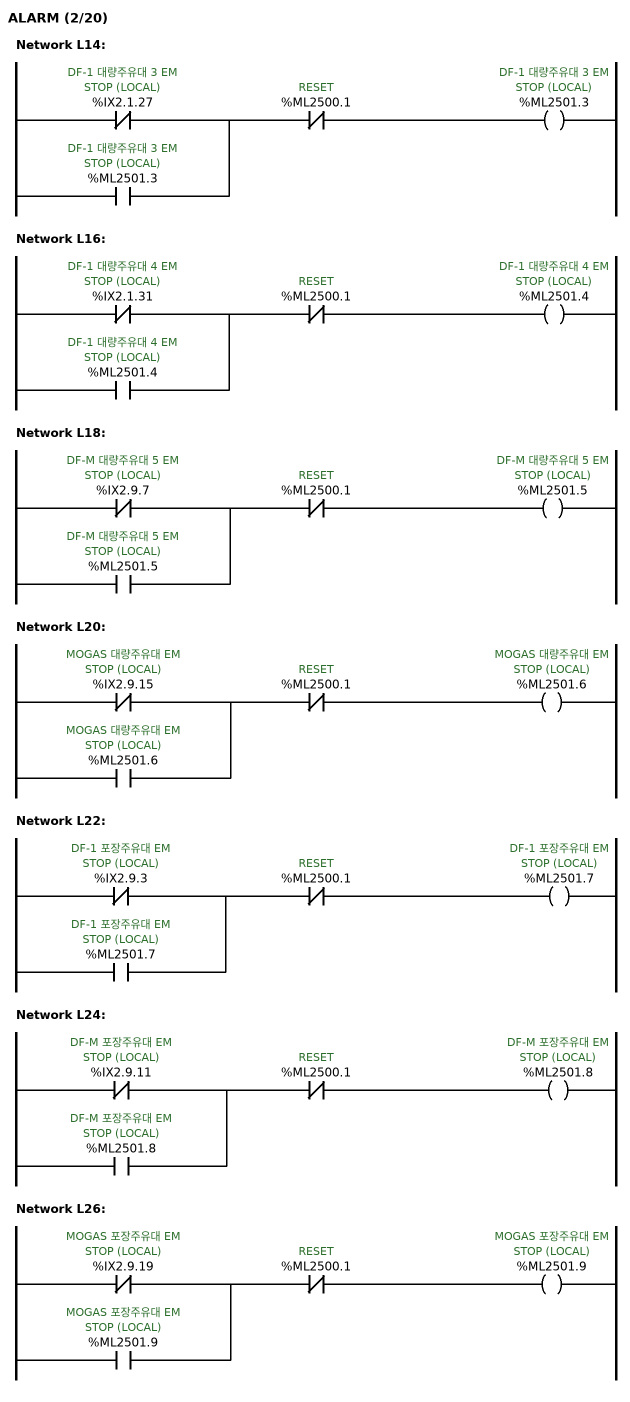
(* Rung L14 *)
%ML2501.3 := (NOT %IX2.1.27 OR %ML2501.3) AND NOT %ML2500.1;
(* Rung L16 *)
%ML2501.4 := (NOT %IX2.1.31 OR %ML2501.4) AND NOT %ML2500.1;
(* Rung L18 *)
%ML2501.5 := (NOT %IX2.9.7 OR %ML2501.5) AND NOT %ML2500.1;
(* Rung L20 *)
%ML2501.6 := (NOT %IX2.9.15 OR %ML2501.6) AND NOT %ML2500.1;
(* Rung L22 *)
%ML2501.7 := (NOT %IX2.9.3 OR %ML2501.7) AND NOT %ML2500.1;
(* Rung L24 *)
%ML2501.8 := (NOT %IX2.9.11 OR %ML2501.8) AND NOT %ML2500.1;
(* Rung L26 *)
%ML2501.9 := (NOT %IX2.9.19 OR %ML2501.9) AND NOT %ML2500.1;

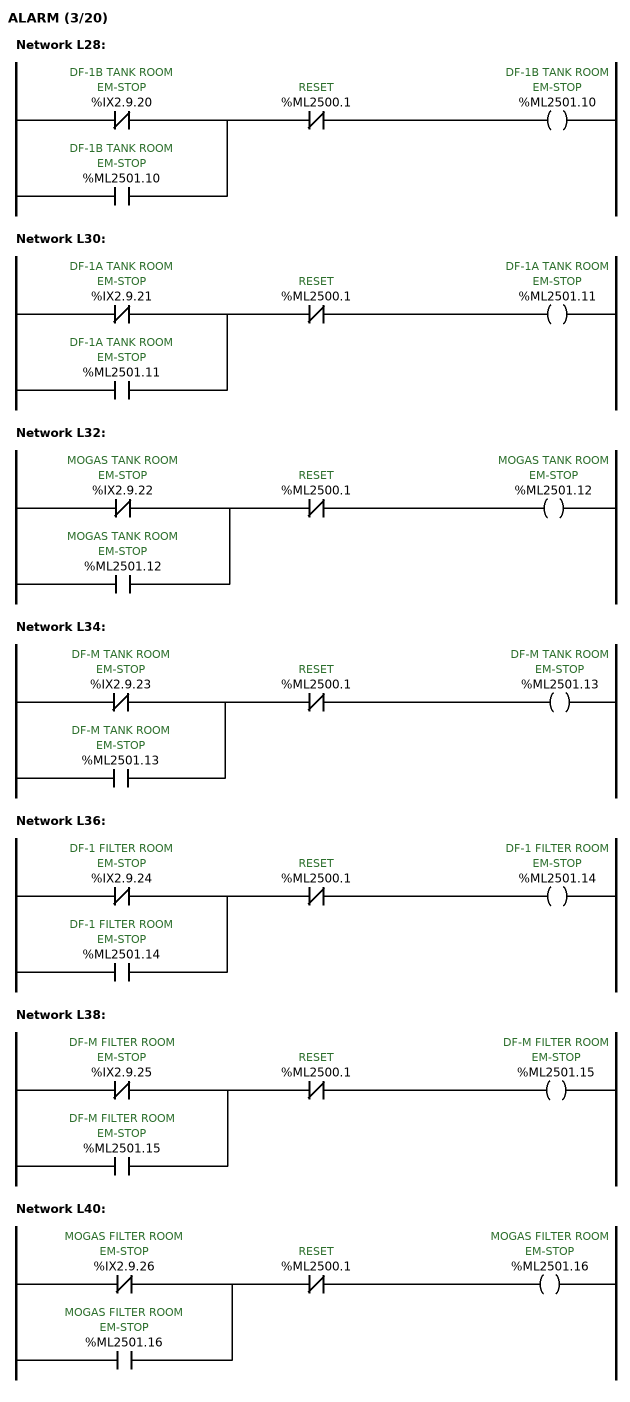
(* Rung L28 *)
%ML2501.10 := (NOT %IX2.9.20 OR %ML2501.10) AND NOT %ML2500.1;
(* Rung L30 *)
%ML2501.11 := (NOT %IX2.9.21 OR %ML2501.11) AND NOT %ML2500.1;
(* Rung L32 *)
%ML2501.12 := (NOT %IX2.9.22 OR %ML2501.12) AND NOT %ML2500.1;
(* Rung L34 *)
%ML2501.13 := (NOT %IX2.9.23 OR %ML2501.13) AND NOT %ML2500.1;
(* Rung L36 *)
%ML2501.14 := (NOT %IX2.9.24 OR %ML2501.14) AND NOT %ML2500.1;
(* Rung L38 *)
%ML2501.15 := (NOT %IX2.9.25 OR %ML2501.15) AND NOT %ML2500.1;
(* Rung L40 *)
%ML2501.16 := (NOT %IX2.9.26 OR %ML2501.16) AND NOT %ML2500.1;

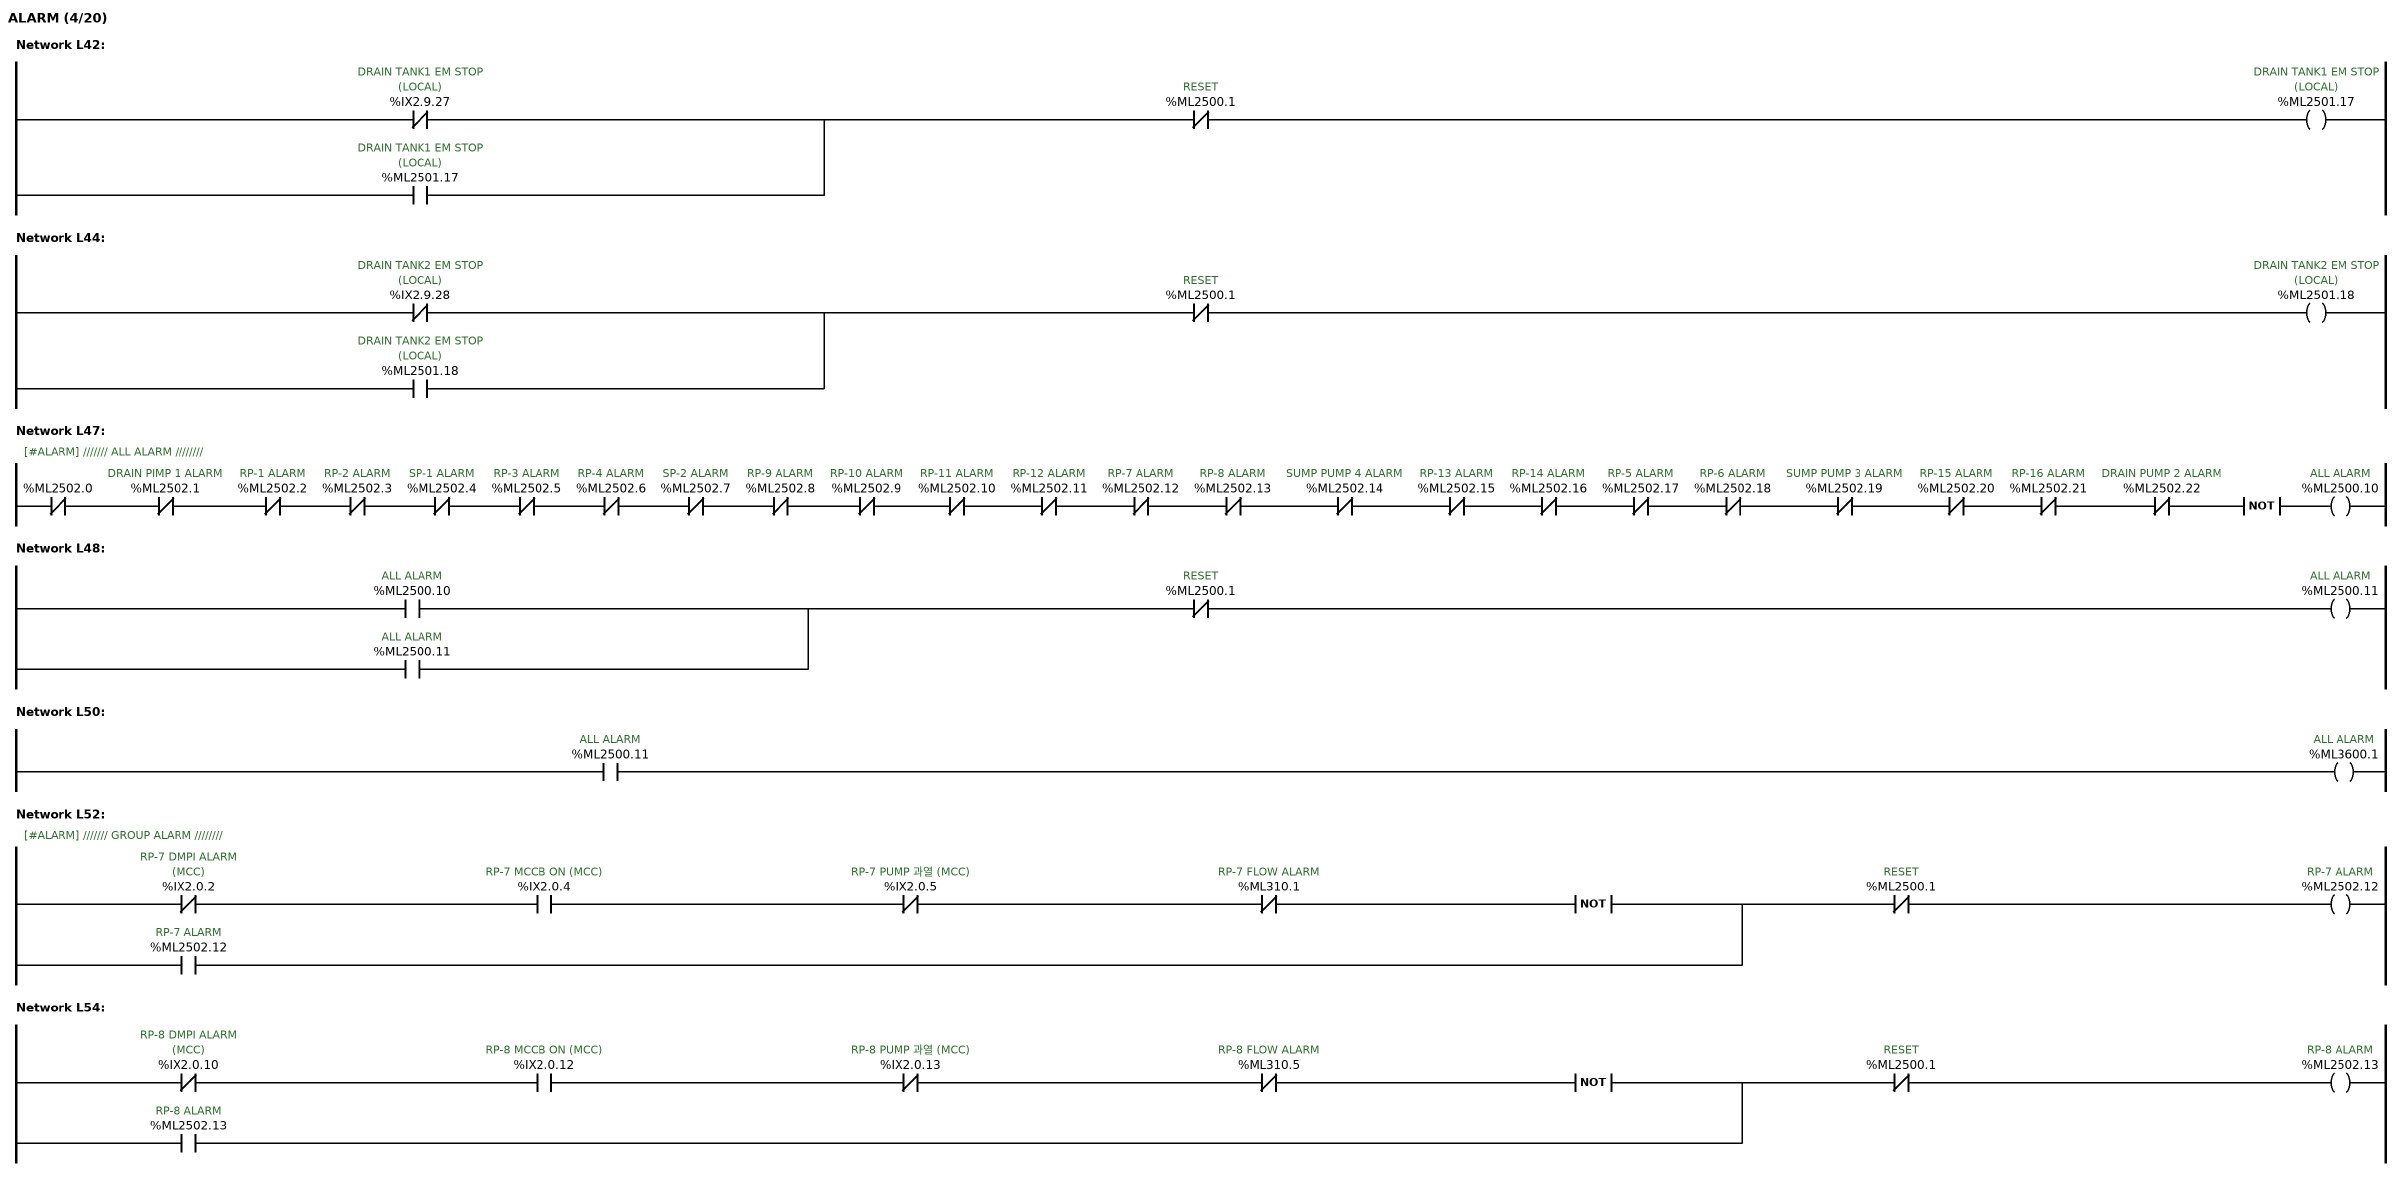
(* Rung L42 *)
%ML2501.17 := (NOT %IX2.9.27 OR %ML2501.17) AND NOT %ML2500.1;
(* Rung L44 *)
%ML2501.18 := (NOT %IX2.9.28 OR %ML2501.18) AND NOT %ML2500.1;
(* [#ALARM] /////// ALL ALARM //////// *)
(* Rung L47 *)
%ML2500.10 := NOT (NOT %ML2502.0 AND NOT %ML2502.1 AND NOT %ML2502.2 AND NOT %ML2502.3 AND NOT %ML2502.4 AND NOT %ML2502.5 AND NOT %ML2502.6 AND NOT %ML2502.7 AND NOT %ML2502.8 AND NOT %ML2502.9 AND NOT %ML2502.10 AND NOT %ML2502.11 AND NOT %ML2502.12 AND NOT %ML2502.13 AND NOT %ML2502.14 AND NOT %ML2502.15 AND NOT %ML2502.16 AND NOT %ML2502.17 AND NOT %ML2502.18 AND NOT %ML2502.19 AND NOT %ML2502.20 AND NOT %ML2502.21 AND NOT %ML2502.22);
(* Rung L48 *)
%ML2500.11 := (%ML2500.10 OR %ML2500.11) AND NOT %ML2500.1;
(* Rung L50 *)
%ML3600.1 := %ML2500.11;
(* [#ALARM] /////// GROUP ALARM //////// *)
(* Rung L52 *)
%ML2502.12 := (NOT (NOT %IX2.0.2 AND %IX2.0.4 AND NOT %IX2.0.5 AND NOT %ML310.1) OR %ML2502.12) AND NOT %ML2500.1;
(* Rung L54 *)
%ML2502.13 := (NOT (NOT %IX2.0.10 AND %IX2.0.12 AND NOT %IX2.0.13 AND NOT %ML310.5) OR %ML2502.13) AND NOT %ML2500.1;

